{attribute 'qualified_only'}
{attribute 'strict'}
TYPE E_MbDevState :
(
	Idle := 0,
	Acquire,
	Wait,
	Cooldown
);
END_TYPE

(* stored: Version 1.1.0.1
   DUT E_MbDevState: Id {fd6e04b1-bb6c-4135-83c2-638e6f9de00f} *)
